# EPICS autosave request: agilent33220A/agilent33220A_settings.req
$(P)$(Q):FREQSTEP
$(P)$(Q):PERFORMRAMP.SCAN
$(P)$(Q):STARTFREQ
$(P)$(Q):STOPFREQ
$(P)$(Q):UPDATE.SCAN
